% RSLogix 500 project INTRO TO PLC - JOB 20.RSS, saved by version 10.00.00.00 %
PROJECT "PL06B"    % processor: Bul.1763 MicroLogix 1100 Series B %

PROGRAM FILES
  LAD 2   12 rungs

DATA FILES
  O0 OUTPUT  4 elements
  I1 INPUT  6 elements
  S2 STATUS  66 elements
  B3 BINARY  1 elements
  T4 TIMER  10 elements
  C5 COUNTER  2 elements
  R6 CONTROL  1 elements
  N7 INTEGER  5 elements
  F8 FLOAT  1 elements

LADDER 2
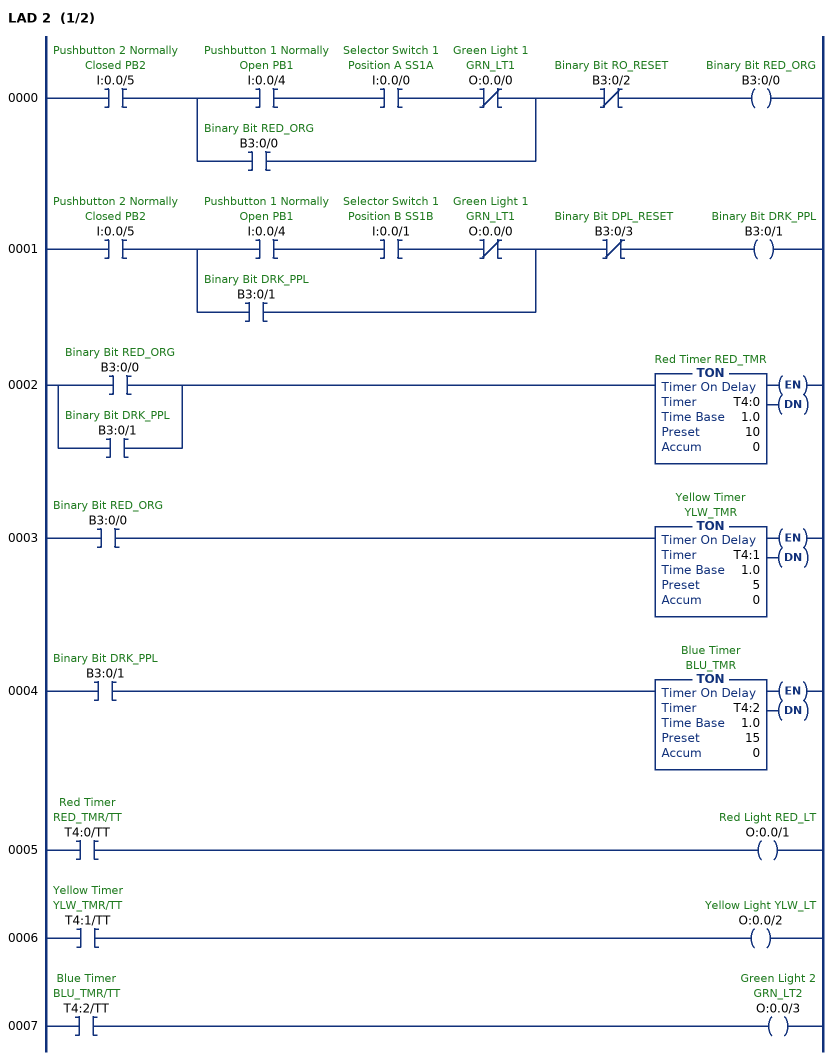
% Rung: 0 %
SOR XIC I:0.0/5 BST XIC I:0.0/4 XIC I:0.0/0 XIO O:0.0/0 NXB XIC B3:0/0 BND XIO B3:0/2 OTE B3:0/0 EOR
%   I:0.0/5  PB2  "Pushbutton 2 Normally Closed" %
%   I:0.0/4  PB1  "Pushbutton 1 Normally Open" %
%   I:0.0/0  SS1A  "Selector Switch 1 Position A" %
%   O:0.0/0  GRN_LT1  "Green Light 1" %
%   B3:0/0  RED_ORG  "Binary Bit" %
%   B3:0/2  RO_RESET  "Binary Bit" %
% Rung: 1 %
SOR XIC I:0.0/5 BST XIC I:0.0/4 XIC I:0.0/1 XIO O:0.0/0 NXB XIC B3:0/1 BND XIO B3:0/3 OTE B3:0/1 EOR
%   I:0.0/5  PB2  "Pushbutton 2 Normally Closed" %
%   I:0.0/4  PB1  "Pushbutton 1 Normally Open" %
%   I:0.0/1  SS1B  "Selector Switch 1 Position B" %
%   O:0.0/0  GRN_LT1  "Green Light 1" %
%   B3:0/1  DRK_PPL  "Binary Bit" %
%   B3:0/3  DPL_RESET  "Binary Bit" %
% Rung: 2 %
SOR BST XIC B3:0/0 NXB XIC B3:0/1 BND TON T4:0 1.0 10 0 EOR
%   B3:0/0  RED_ORG  "Binary Bit" %
%   B3:0/1  DRK_PPL  "Binary Bit" %
%   T4:0  RED_TMR  "Red Timer" %
% Rung: 3 %
SOR XIC B3:0/0 TON T4:1 1.0 5 0 EOR
%   B3:0/0  RED_ORG  "Binary Bit" %
%   T4:1  YLW_TMR  "Yellow Timer" %
% Rung: 4 %
SOR XIC B3:0/1 TON T4:2 1.0 15 0 EOR
%   B3:0/1  DRK_PPL  "Binary Bit" %
%   T4:2  BLU_TMR  "Blue Timer" %
% Rung: 5 %
SOR XIC T4:0/TT OTE O:0.0/1 EOR
%   T4:0  RED_TMR  "Red Timer" %
%   O:0.0/1  RED_LT  "Red Light" %
% Rung: 6 %
SOR XIC T4:1/TT OTE O:0.0/2 EOR
%   T4:1  YLW_TMR  "Yellow Timer" %
%   O:0.0/2  YLW_LT  "Yellow Light" %
% Rung: 7 %
SOR XIC T4:2/TT OTE O:0.0/3 EOR
%   T4:2  BLU_TMR  "Blue Timer" %
%   O:0.0/3  GRN_LT2  "Green Light 2" %

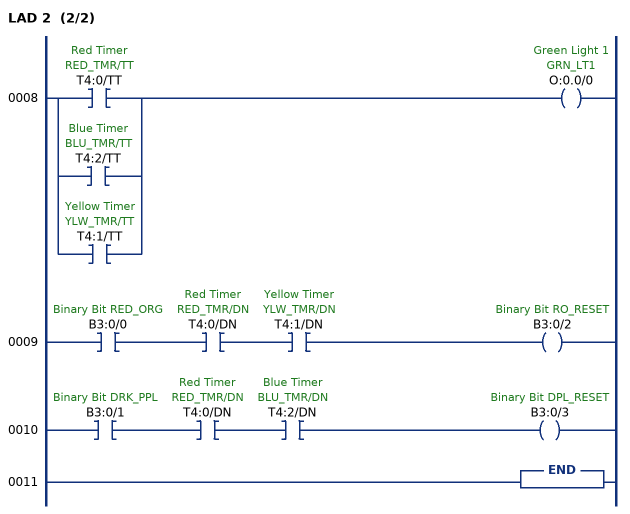
% Rung: 8 %
SOR BST XIC T4:0/TT NXB XIC T4:2/TT NXB XIC T4:1/TT BND OTE O:0.0/0 EOR
%   T4:0  RED_TMR  "Red Timer" %
%   T4:2  BLU_TMR  "Blue Timer" %
%   T4:1  YLW_TMR  "Yellow Timer" %
%   O:0.0/0  GRN_LT1  "Green Light 1" %
% Rung: 9 %
SOR XIC B3:0/0 XIC T4:0/DN XIC T4:1/DN OTE B3:0/2 EOR
%   B3:0/0  RED_ORG  "Binary Bit" %
%   T4:0  RED_TMR  "Red Timer" %
%   T4:1  YLW_TMR  "Yellow Timer" %
%   B3:0/2  RO_RESET  "Binary Bit" %
% Rung: 10 %
SOR XIC B3:0/1 XIC T4:0/DN XIC T4:2/DN OTE B3:0/3 EOR
%   B3:0/1  DRK_PPL  "Binary Bit" %
%   T4:0  RED_TMR  "Red Timer" %
%   T4:2  BLU_TMR  "Blue Timer" %
%   B3:0/3  DPL_RESET  "Binary Bit" %
% Rung: 11 %
SOR END EOR

OTHER DOCUMENTED ADDRESSES
  B3:0/4  GRN_STOP  "Green Light 1 Stop"
  B3:0/15  SCRATCH  "Scratch Bit"
  B3:1/1  RED_TMR_DNS  "Red Light Timer Done Storage"
  C5:0  FLR1_CTR  "First Floor Counter"
  C5:1  FLR2_CTR  "Second Floor Counter"
  I  
  I:0.0/2  SS2A  "Selector Switch 2 Position A"
  I:0.0/3  SS2B  "Selector Switch 2 Position B"
  RTC:0.YR  RTC
  SEL1B  
  T4:3  RST_TMR  "Reset Timer"

DATA TABLE (non-zero values as saved)
DATA B3
% B3:0 % 0X8009
DATA T4
% .PRE .ACC %
% T4:0 % 10 0
% T4:1 % 5 0
% T4:2 % 15 0
% T4:3 % 10 0
DATA C5
% .PRE .ACC %
% C5:1 % 0 10
DATA N7
% N7:0 % 555 0 0 0 0
